FUNCTION_BLOCK FB_SetEnables_Test EXTENDS TcUnit.FB_TestSuite
VAR
    Expected: BOOL := True;
    Actual: BOOL;
END_VAR

TEST('FB_SetEnables_Test Dummy Test');
AssertEquals(Expected := Expected,
             Actual := Actual,
             Message := 'Error Message');
TEST_FINISHED();

END_FUNCTION_BLOCK

(* stored: Version 1.1.0.1, ProductVersion 3.1.4022.18
   POU FB_SetEnables_Test: Id {fa7a8f28-80a8-4902-a8cc-143983714ddb}, SpecialFunc None *)
